PROGRAM IOLink
VAR


	Spare: BOOL;

	TiersheetRemoverUP: SR;
	SheetRemoverUP: BOOL;
	TiersheetCarriage_Auto: BOOL;
	Remove_Dn_TMR: TON;
END_VAR

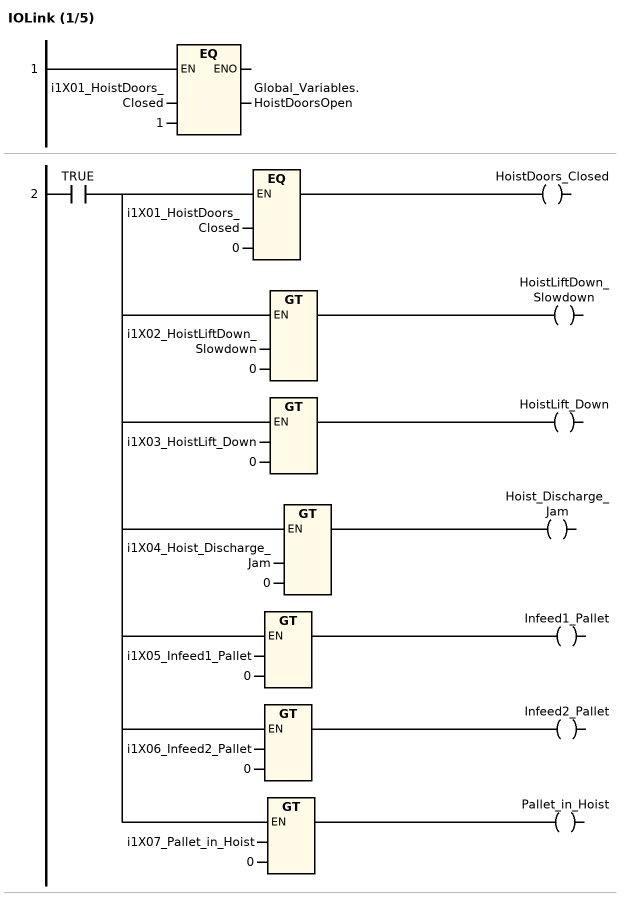
// NETWORK 1
Global_Variables.HoistDoorsOpen := i1X01_HoistDoors_Closed = 1;

// NETWORK 2
HoistDoors_Closed := i1X01_HoistDoors_Closed = 0;
HoistLiftDown_Slowdown := i1X02_HoistLiftDown_Slowdown > 0;
HoistLift_Down := i1X03_HoistLift_Down > 0;
Hoist_Discharge_Jam := i1X04_Hoist_Discharge_Jam > 0;
Infeed1_Pallet := i1X05_Infeed1_Pallet > 0;
Infeed2_Pallet := i1X06_Infeed2_Pallet > 0;
Pallet_in_Hoist := i1X07_Pallet_in_Hoist > 0;

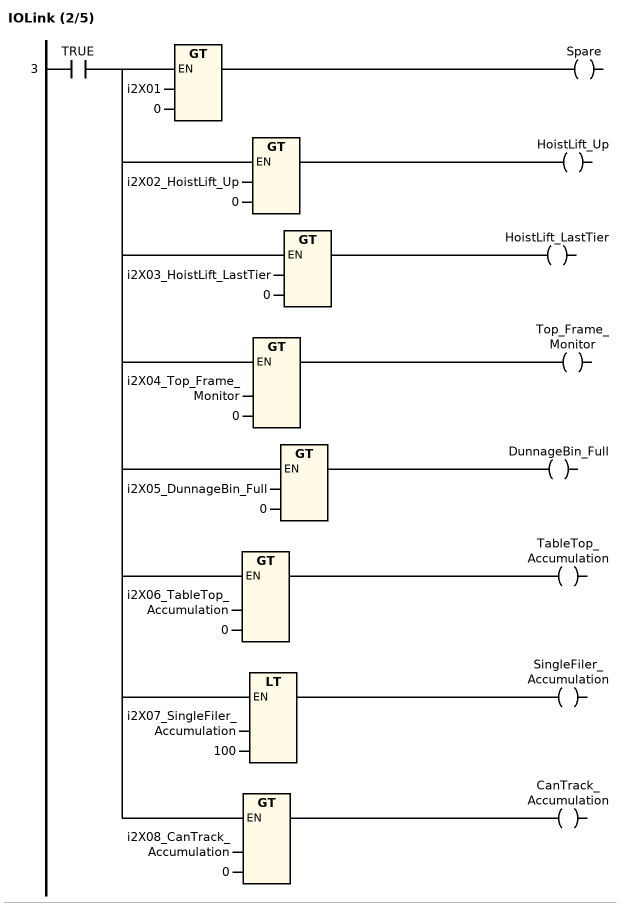
// NETWORK 3
Spare := i2X01 > 0;
HoistLift_Up := i2X02_HoistLift_Up > 0;
HoistLift_LastTier := i2X03_HoistLift_LastTier > 0;
Top_Frame_Monitor := i2X04_Top_Frame_Monitor > 0;
DunnageBin_Full := i2X05_DunnageBin_Full > 0;
TableTop_Accumulation := i2X06_TableTop_Accumulation > 0;
SingleFiler_Accumulation := i2X07_SingleFiler_Accumulation < 100;
CanTrack_Accumulation := i2X08_CanTrack_Accumulation > 0;

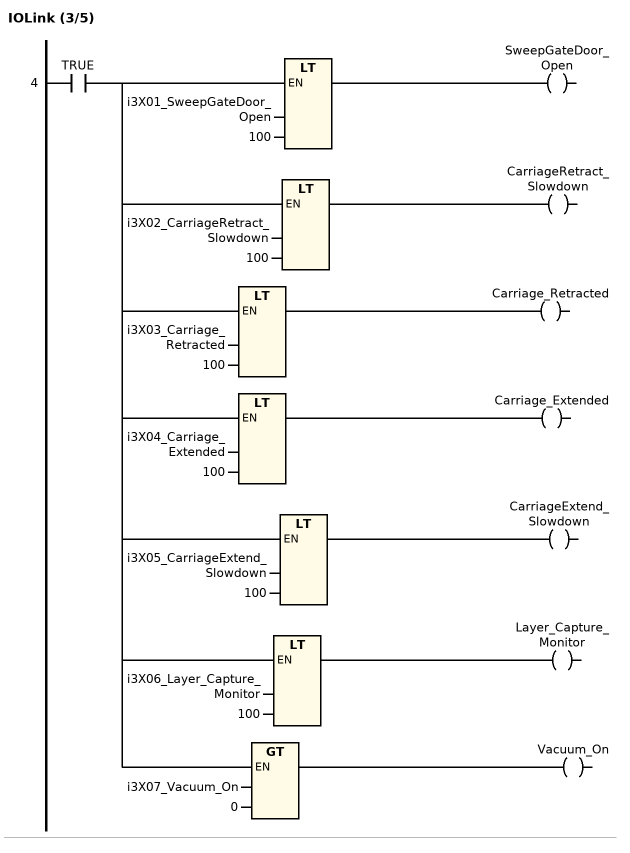
// NETWORK 4
SweepGateDoor_Open := i3X01_SweepGateDoor_Open < 100;
CarriageRetract_Slowdown := i3X02_CarriageRetract_Slowdown < 100;
Carriage_Retracted := i3X03_Carriage_Retracted < 100;
Carriage_Extended := i3X04_Carriage_Extended < 100;
CarriageExtend_Slowdown := i3X05_CarriageExtend_Slowdown < 100;
Layer_Capture_Monitor := i3X06_Layer_Capture_Monitor < 100;
Vacuum_On := i3X07_Vacuum_On > 0;

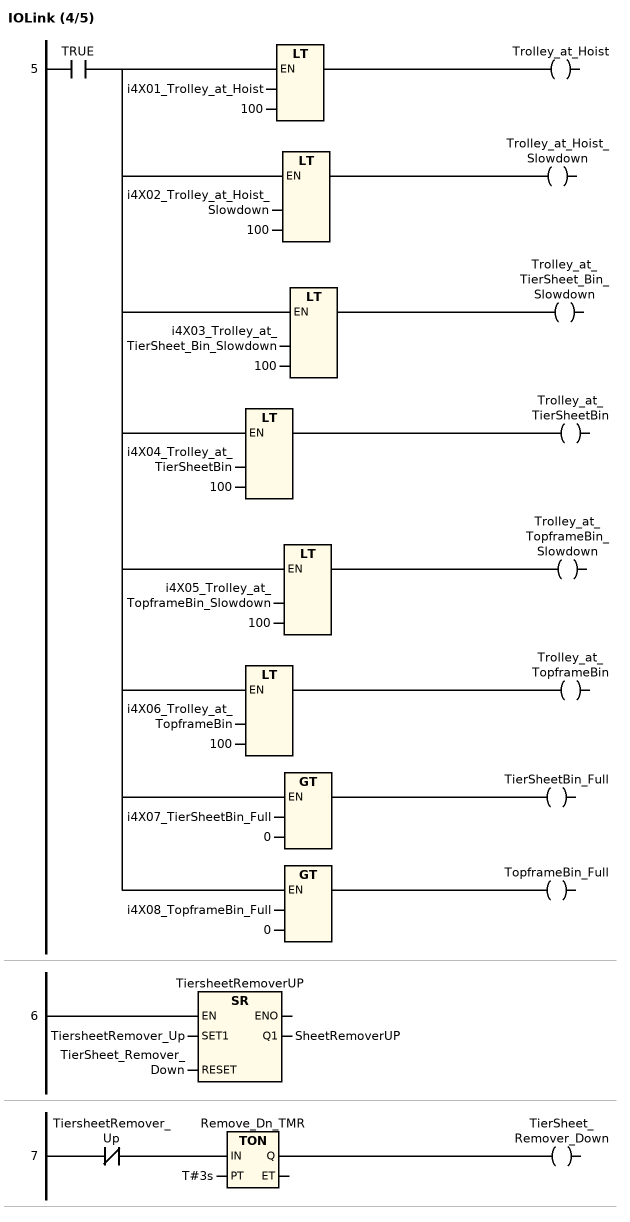
// NETWORK 5
Trolley_at_Hoist := i4X01_Trolley_at_Hoist < 100;
Trolley_at_Hoist_Slowdown := i4X02_Trolley_at_Hoist_Slowdown < 100;
Trolley_at_TierSheet_Bin_Slowdown := i4X03_Trolley_at_TierSheet_Bin_Slowdown < 100;
Trolley_at_TierSheetBin := i4X04_Trolley_at_TierSheetBin < 100;
Trolley_at_TopframeBin_Slowdown := i4X05_Trolley_at_TopframeBin_Slowdown < 100;
Trolley_at_TopframeBin := i4X06_Trolley_at_TopframeBin < 100;
TierSheetBin_Full := i4X07_TierSheetBin_Full > 0;
TopframeBin_Full := i4X08_TopframeBin_Full > 0;

// NETWORK 6
TiersheetRemoverUP(SET1 := TiersheetRemover_Up, RESET := TierSheet_Remover_Down, Q1 => SheetRemoverUP); // SR

// NETWORK 7
Remove_Dn_TMR(IN := NOT TiersheetRemover_Up, PT := T#3s); // TON
TierSheet_Remover_Down := Remove_Dn_TMR.Q;

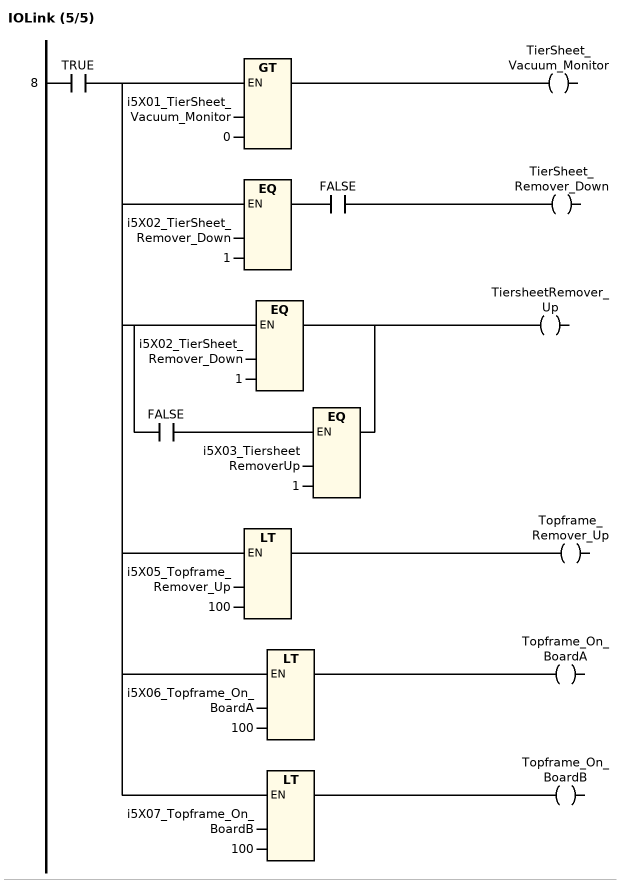
// NETWORK 8
TierSheet_Vacuum_Monitor := i5X01_TierSheet_Vacuum_Monitor > 0;
TierSheet_Remover_Down := i5X02_TierSheet_Remover_Down = 1 AND FALSE;
TiersheetRemover_Up := i5X02_TierSheet_Remover_Down = 1 OR TRUE AND FALSE AND i5X03_TiersheetRemoverUp = 1;
Topframe_Remover_Up := i5X05_Topframe_Remover_Up < 100;
Topframe_On_BoardA := i5X06_Topframe_On_BoardA < 100;
Topframe_On_BoardB := i5X07_Topframe_On_BoardB < 100;

END_PROGRAM

(* stored: Version 1.1.0.1, ProductVersion 3.1.4024.16
   POU IOLink: Id {6171b43c-9a3a-45f4-ad83-db32b5ae9c89}, SpecialFunc None *)
